// TIA Portal V18 export
DATA_BLOCK "05_EM_STATE"   // DB7, F_DB
{ S7_Optimized_Access := 'TRUE'; DB_Accessible_From_OPC_UA := 'FALSE' }
// stored: DBAccessibleFromOPCUA false
   VAR
      "Always FALSE" : Bool;
      "Always TRUE" : Bool := TRUE;
      RESET : Bool;
      "!!05_EM_STATE.{matrix_area}_SORTER_NOT_RUNNING$$" : Bool;
      "!!05_EM_STATE.{matrix_area}_SORTER_POWER_CUT$$" : Bool;
      "!!05_EM_STATE.{matrix_area}_SAFETY_DOORS_COM$$" : Bool;
      "!!05_EM_STATE.{matrix_area}_SAFETY_BREAKERS_COM$$" : Bool;
      "!!05_EM_STATE.{matrix_area}_Q$$" : Bool;
      "!!05_EM_STATE.{matrix_area}_Q_DELAYED$$" : Bool;
      "!!05_EM_STATE.{matrix_areas.1}$$" : Bool;
      "!!05_EM_STATE.{matrix_areas.2}$$" : Bool;
      "!!05_EM_STATE.{matrix_areas.3}$$" : Bool;
      "!!05_EM_STATE.{matrix_areas.4}$$" : Bool;
      "!!05_EM_STATE.{matrix_areas.1}_RESET$$" : Bool;
      "!!05_EM_STATE.{matrix_areas.2}_RESET$$" : Bool;
      "!!05_EM_STATE.{matrix_areas.3}_RESET$$" : Bool;
      "!!05_EM_STATE.{matrix_areas.4}_RESET$$" : Bool;
   END_VAR
BEGIN
END_DATA_BLOCK
